KUKA KRL program: LAB_OL_KR3.src, LAB_OL_KR3.dat

--- LAB_OL_KR3.src ---
&ACCESS RVP
&REL 1
&PARAM TEMPLATE = C:\KRC\Roboter\Template\vorgabe
&PARAM EDITMASK = *
DEF LAB_OL_KR3()
  ; KLAB fixture: isolated OfficeLite KR3 bounded execution only
  BAS(#INITMOV,0)
  $ADVANCE=0
  $IPO_MODE=#BASE
  $ORI_TYPE=#VAR
  BAS(#TOOL,0)
  BAS(#BASE,0)
  $ACC.CP=1.0
  $VEL.ORI1=100
  $VEL.ORI2=100
  $ACC.ORI1=100
  $ACC.ORI2=100
  $APO.CDIS=0
  $APO.CPTP=0
  BAS(#VEL_PTP,20)
  BAS(#ACC_PTP,20)
  PTP A_HOME
  $VEL.CP=0.05
  LIN_REL P_DELTA
END

--- LAB_OL_KR3.dat ---
&ACCESS RVP
&REL 1
DEFDAT LAB_OL_KR3 PUBLIC
  DECL E6AXIS A_HOME={A1 0,A2 -90,A3 90,A4 0,A5 0,A6 0,E1 0,E2 0,E3 0,E4 0,E5 0,E6 0}
  DECL FRAME P_DELTA={X 10,Y 0,Z 0,A 0,B 0,C 0}
ENDDAT
